# EPICS autosave request: measCompApp/Db/C9513_pulse_generator_settings.req
$(P)$(R)PulsePeriod
$(P)$(R)PulseWidth
$(P)$(R)PulseDelay
$(P)$(R)PulseIdleState
$(P)$(R)PulseCount
